TYPE Loader :
STRUCT
	Level_Prox AT%I* : BOOL;
	Flap_Reed AT%I* : BOOL;
	Switch AT%I* : BOOL;
	PushButton AT%I* : BOOL;
	Valve AT%Q* : BOOL;
	Lamp AT%Q* : BOOL;
	Status_Word : WORD;
	HMI_Status_Word : WORD;
END_STRUCT
END_TYPE

(* stored: Version 1.1.0.1, ProductVersion 3.1.4024.13
   DUT Loader: Id {8c85dd9f-7832-4bf7-9976-9ace8fcebe8b} *)
